RoboDK station: UR3e mit Robotiq First Test Camera.rdk

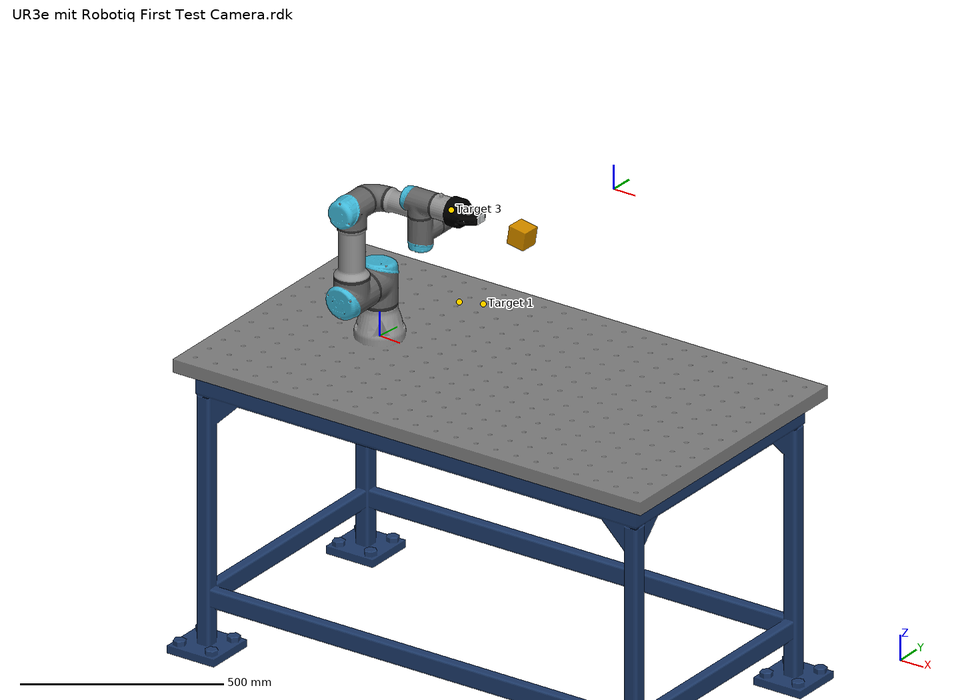
[picture v0: the station drawn from its stored meshes, robots at their saved joint values, targets as dots, program paths as lines]
Station UR3e mit Robotiq First Test Camera (saved by RoboDK 5.9.5). Poses are relative to the parent item; angles as X-Y-Z fixed-axis rotations.
Station parameters (name, value as stored): OPC-UA, opc.tcp://localhost:4840
  - frame UR3e Base at (0, 0, 0) mm, rotated rx 0 ry 0 rz -6.26 deg
    - robot UR3e: 6 axes, payload 3 kg, reach 500 mm, repeatability 0.03 mm, weight 11 kg
        modified DH rows (alpha deg, a mm, theta deg, d mm): 0, 0, 0, 151.9; 90, 0, 180, 0; 0, 243.55, 0, 0; 0, 213.2, 0, 131.05; -90, 0, 0, 85.35; 90, 0, 180, 92.1
        joint limits [-360, -360, -360, -360, -360, -360] to [360, 360, 360, 360, 360, 360]; home [0, -90, -90, 0, 90, 0]; saved at [6.26, -90.001, -90.429, 0.431, 90, 0]
      - robot RobotiQ 2F-85 Gripper (Mechanism) (model RobotiQ 2F85): 1 axes, payload 5 kg
          joint limits [0] to [85]; home [85]; saved at [85]
        - tool Tool 1, TCP at (0, 0, 160) mm
  - object Table 1400x800x800mm at (0, 0, 0) mm, size 1420 x 820 x 800 mm, geometry from Table-1400x800x800mm.sld
    - object Cube 50mm at (326.81, -143.51, 0) mm, rotated rx 0 ry -78.13 rz 0 deg, size 50 x 50 x 50 mm, geometry from Cube-50mm.sld
    - object Intel RealSense D435 Camera at (0, 0, 2000) mm, rotated rx 180 ry 0 rz 0 deg, size 89.8 x 25 x 25.1 mm, geometry from Intel-RealSense-D435-Camera.sld
  - frame RobotiQ 2F-85 Gripper (Mechanism) Base at (0, 1000, 0) mm
    - target Target 1 (Cartesian target) at (401.23, -1130.82, 250.26) mm, rotated rx 108.04 ry 86.9 rz -161.94 deg; joints [140.623, 11.663, -29.078, -163.926, 45.694, 93.884] of UR3e
    - target Target 3 (Cartesian target) at (305.3, -1131.05, 479.2) mm, rotated rx -90 ry 0 rz -90 deg; joints [6.26, -90.001, -90.429, 0.431, 90, 0] of UR3e
    - target Target 2 (Cartesian target) at (329.51, -1131.05, 236.31) mm, rotated rx 177.05 ry 1.7 rz -90.09 deg; joints [5.792, -100.67, -95.278, -77.012, 91.677, -0.468] of UR3e
  - Python program Prog_Attach (listed below)
  - Python program Prog_Camera (listed below)
  - frame RGB Camera Frame at (300, -40, 1200) mm, rotated rx 180 ry 0 rz 0 deg
  - camera My Camera
  - Python program Prog_Depth_Cam (listed below)
  - camera Depth Camera
  - camera Intel RealSense D435 Camera
  - frame RealsenseCamFrame at (534.87, -28.09, 3000) mm, rotated rx -176.51 ry -1.78 rz 180 deg

--- Python program Prog_Attach ---
# This script allows you to attach an object to a robot link
# https://robodk.com/doc/en/PythonAPI/examples.html#attach-object-to-a-robot-link

from robodk.robolink import *  # API to communicate with RoboDK
from robodk.robodialogs import *

RDK = Robolink()  # Initialize the RoboDK API

# Select the robot
# Add the shape to a robot link
robot = RDK.ItemUserPick('Select a robot to add an object', ITEM_TYPE_ROBOT)
if not robot.Valid():
    raise Exception('No robot selected. Add a robot to attach this geometry to a link')

while True:
    value = mbox('Enter the joint to attach the object to:\n' + robot.Name() + '\nExample: 0 is the base, 3 is joint 3', entry='3')
    if not value:
        quit(0)

    link_id = int(value)
    robotlink = robot.ObjectLink(link_id)
    if robotlink.Valid():
        break

    RDK.ShowMessage("Invalid link. Select a valid robot link")

object = RDK.ItemUserPick('Select the object to add', ITEM_TYPE_OBJECT)
if not object.Valid():
    raise Exception('Object not selected')

# List of objects to merge (first one must be the robot link)
merge = [robotlink, object]

# Merge the object
RDK.MergeItems(merge)

# Set original object invisible (or delete)
object.setVisible(False)
# object.Delete()

--- Python program Prog_Camera ---
# Type help("robodk.robolink") or help("robodk.robomath") for more information
# Press F5 to run the script
# Documentation: https://robodk.com/doc/en/RoboDK-API.html
# Reference:     https://robodk.com/doc/en/PythonAPI/index.html
#
# This example demonstrates some of the basic functionalities to handle 2D cameras using the RoboDK API for Python.
# It creates/reuses an existing camera, set its parameters, get the image using two different methods and display it to the user as a live stream.
# This is a great starting point for your computer vision algorithms.
#

from robodk import robolink  # RoboDK API
from robodk import robomath  # Robot toolbox
RDK = robolink.Robolink()

# OpenCV is an open source Computer Vision toolkit, which you can use to filter and analyse images
# https://robodk.com/doc/en/PythonAPI/examples.html#camera-2d
robolink.import_install('cv2', 'opencv-python', RDK)
robolink.import_install('numpy', RDK)
import numpy as np
import cv2 as cv

CAM_NAME = 'My Camera'
CAM_PARAMS = 'SIZE=640x480' # For more options, see https://robodk.com/doc/en/PythonAPI/robodk.html#robodk.robolink.Robolink.Cam2D_Add
WINDOW_NAME = 'My Camera Feed'

#----------------------------------
# Get the camera item
cam_item = RDK.Item(CAM_NAME, robolink.ITEM_TYPE_CAMERA)
if not cam_item.Valid():
    cam_item = RDK.Cam2D_Add(RDK.AddFrame(CAM_NAME + ' Frame'), CAM_PARAMS)
    cam_item.setName(CAM_NAME)
cam_item.setParam('Open', 1)

#----------------------------------
# Create a live feed
while cam_item.setParam('isOpen') == '1':

    #----------------------------------
    # Method 1: Get the camera image, by socket
    img_socket = None
    bytes_img = RDK.Cam2D_Snapshot('', cam_item)
    if isinstance(bytes_img, bytes) and bytes_img != b'':
        nparr = np.frombuffer(bytes_img, np.uint8)
        img_socket = cv.imdecode(nparr, cv.IMREAD_COLOR)
    if img_socket is None:
        break

    #----------------------------------
    # Method 2: Get the camera image, from disk
    img_png = None
    import tempfile
    with tempfile.TemporaryDirectory(prefix='robodk_') as td:
        tf = td + '/temp.png'
        if RDK.Cam2D_Snapshot(tf, cam_item) == 1:
            img_png = cv.imread(tf)
    if img_png is None:
        break

    #----------------------------------
    # Show it to the world!
    cv.imshow(WINDOW_NAME, img_socket)
    key = cv.waitKey(1)
    if key == 27:
        break  # User pressed ESC, exit
    if cv.getWindowProperty(WINDOW_NAME, cv.WND_PROP_VISIBLE) < 1:
        break  # User killed the main window, exit

# Close the preview and the camera. Ensure you call cam_item.setParam('Open', 1) before reusing a camera!
cv.destroyAllWindows()
RDK.Cam2D_Close(cam_item)

--- Python program Prog_Depth_Cam ---
# https://robodk.com/doc/en/PythonAPI/examples.html#depth-camera-3d
# Type help("robolink") or help("robodk") for more information
# Press F5 to run the script
# Documentation: https://robodk.com/doc/en/RoboDK-API.html
# Reference:     https://robodk.com/doc/en/PythonAPI/index.html
#
# This example shows how to retrieve and display the 32-bit depth map of a simulated camera.

from robodk.robolink import *  # RoboDK API

from tempfile import TemporaryDirectory
import numpy as np
from matplotlib import pyplot as plt

#----------------------------------
# Get the simulated camera from RoboDK
RDK = Robolink()

# existierende Kamera holen oder neu anlegen
cam_item = RDK.Item('Intel RealSense D435 Camera', ITEM_TYPE_CAMERA)
if not cam_item.Valid():
    cam_item = RDK.Cam2D_Add(
        RDK.ActiveStation(),
        'SIZE=160x160 SNAPSHOT=160x160 FAR_LENGTH=120 DEPTH'
    )
    cam_item.setName('Intel RealSense D435 Camera')

cam_item.setParam('Open', 1)
#----------------------------------------------
# Get the image from RoboDK
td = TemporaryDirectory(prefix='robodk_')
tf = td.name + '/temp.grey32'
if RDK.Cam2D_Snapshot(tf, cam_item) == 1:
    grey32 = np.fromfile(tf, dtype='>u4')
    if grey32.size < 2:
        raise RuntimeError("Depth file too small, no data written")
    w, h = grey32[:2]
    if grey32.size != 2 + w * h:
        raise RuntimeError(f"Depth size mismatch: got {grey32.size}, expected {2 + w*h}")
    grey32 = np.flipud(np.reshape(grey32[2:], (h, w)))
else:
    raise RuntimeError("Cam2D_Snapshot failed")

#----------------------------------------------
# Display
grey32[grey32 == 0] = 2**32 - 1  # This is for display purposes only! Values of 0 do not have any measurements.
plt.imshow(grey32, 'gray')
plt.show()
